Staubli VAL3: clkPark2.pgx

program clkPark2()
begin
  // -- inconsistent implementation compared to clkPark1 and park1 :-)
  call setSpeed()
  resetMotion()
  movej(jInitialPosition, tTool, mFast)
  waitEndMove()
end
